FUNCTION_BLOCK mainGUIFB (* JADE WORKER *)
  (* Standard: 61499-1 *)
  (* Version 1.0, 2014-04-22, Ahmed, Fraunhofer IGD *)
  (* Compiler header: package fb.rt; *)
  (* Compiler Java Sun JDK 1.5.0 *)
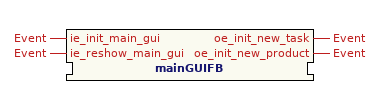
  EVENT_INPUT
    ie_init_main_gui;
    ie_reshow_main_gui;
  END_EVENT
  EVENT_OUTPUT
    oe_init_new_task;
    oe_init_new_product;
  END_EVENT
END_FUNCTION_BLOCK
